Fanuc KAREL source: kt00539.KL

-- PROVISIONAL review KL for V1013-1; original PC SHA256 697ce5afb8317dcb5bc543ce05c619f7b1f721244f0d3649561342e1ee803350
-- Incomplete behavior may be omitted. Consult companion uncertainty JSON. Do not deploy.
PROGRAM KT00539
%NOLOCKGROUP
-- UNRESOLVED_DECL P1 type=000199
-- UNRESOLVED_DECL P2 type=000102
-- UNRESOLVED_DECL OUT type=000101
BEGIN
  -- UNRESOLVED_PC offsets 5-20; opcodes 2E,22,32,35
  -- UNRESOLVED_PC offsets 25-59; opcodes 49,7E,49,7E,60,4A
  -- UNRESOLVED_PC offsets 64-68; opcodes 7F
END KT00539
